// Provide logging 
FUNCTION_BLOCK FB_FileLogging IMPLEMENTS I_Logging
VAR_INPUT
	eLogLevel:				E_LogLevel:= E_LogLevel.Verbose;
END_VAR
VAR_OUTPUT
END_VAR
VAR
	iLogging:				I_Logging;
END_VAR

METHOD PUBLIC M_Attach : BOOL
VAR_INPUT
	iLogging:				I_Logging;
END_VAR
IF THIS^.iLogging = 0 THEN
	THIS^.iLogging:= iLogging;
	M_Attach:= TRUE;
ELSIF THIS^.iLogging = iLogging THEN
	// already inside
	M_Attach:= TRUE;
	RETURN;
ELSE
	// redirect to next logging function block
	THIS^.iLogging.M_Attach(iLogging);
END_IF
END_METHOD

METHOD PUBLIC M_Log : BOOL
VAR_INPUT
	stMessage:			ST_Message;
END_VAR
END_METHOD

PROPERTY PUBLIC P_LogLevel : E_LogLevel
GET
P_LogLevel:= eLogLevel;
END_GET
SET
eLogLevel:= P_LogLevel;
END_SET
END_PROPERTY

END_FUNCTION_BLOCK

(* stored: Version 1.1.0.1
   POU FB_FileLogging: Id {9a6a3514-7dcc-42ca-8394-f112c0e45419}, SpecialFunc None
   Method M_Attach: Id {0027130b-1adf-4ef8-b1b0-509d54331a0c}
   Method M_Log: Id {757dfb5f-b25f-4a7d-b4b5-e64d3c75e129}
   Property P_LogLevel: Id {3c08d044-f3e7-4900-b273-c5b3e4af3b4d}
   Get Get: Id {08e69a52-2a9b-4b9b-a4dc-4ef57f155340}
   Set Set: Id {b480e56f-e4d1-407c-b08a-38e5017c1aca} *)
